{attribute 'qualified_only'}
VAR_GLOBAL
	g_CPPTestVar:LREAL;
END_VAR

(* stored: Version 1.1.0.1, ProductVersion 3.1.4024.12
   GVL GVL_CPPTest: Id {99054502-19ce-451a-a908-196cc10c2b5e} *)
